// TIA Portal project "TP2 [A2182]" (V20)

(* hardware
DEVICE "S7-1200 station_1"  S7-1200 Station
   slot 0: "Rack_0"  S7-1200 Rack  Rack  V1.0
   slot 1: "PLC_1"  CPU 1215C DC/DC/Rly  6ES7 215-1HG40-0XB0  V4.2
DEVICE "SINAMICS G_1"  Sinamics.Device
   slot 0: "	_0"  Rail  SinamicsG120SVecto
   slot 0: "Drive_1"  G120 CU250S-2 PN Vector  6SL3246-0BA22-1FA0  4.7.6
      slot 1: "PROFINET interface"  MDD-SinamicsG120-P
   slot 3: "PM240-2 IP20"  PM240-2 IP20  6SL3210-1PB13-8ULx  -
DEVICE "HMI_1"  KTP700 Basic PN
   slot 0: "HMI_1"  KTP700 Basic PN  6AV2 123-2GB03-0AX0  17.0.0.0
   slot 1: "HMI_RT_1"  KTP700 Basic PN  6AV2 123-2GB03-0AX0  17.0.0.0
   slot 5: "HMI_1.IE_CP_1"  PROFINET Interface  17.0.0.0
      slot 1: "PROFINET Interface_1"  PROFINET Interface
         slot 1: "Port_1"  Port
*)

// ===== PLC "PLC_1"  CPU 1215C DC/DC/Rly =====

VAR_GLOBAL   // PLC tag table "Variateur"
   "Ix_EquartVitesse" AT %I500.0 : Bool;   // True = Dans la tolérance, OK
   "Ix_CommandeDemandé" AT %I500.1 : Bool;   // True = OK
   "Ix_VitesseAtteinte" AT %I500.2 : Bool;   // True = Atteint
   "Ix_LimiteCouple" AT %I500.3 : Bool;   // True = Couple Atteint
   "Ix_Frein" AT %I500.4 : Bool;   // True =Freiné
   "Ix_AlarmeSurchauffe" AT %I500.5 : Bool;   // True = OK
   "Ix_RotationDroite" AT %I500.6 : Bool;   // True = Droite
   "Ix_SurchauffeVariateur" AT %I500.7 : Bool;   // True = OK
   "Ix_PretEnclanchement" AT %I501.0 : Bool;   // True = Pret
   "Ix_MoteurTourne" AT %I501.1 : Bool;   // True = Moteur ON
   "Ix_FonctionnementDébloqué" AT %I501.2 : Bool;   // True = OK
   "Ix_DéfautActif" AT %I501.3 : Bool;   // True = Défauts
   "Ix_Arret2innactif" AT %I501.4 : Bool;   // True = Désactivé
   "Ix_Arret3innactif" AT %I501.5 : Bool;   // True = Désactivé
   "Ix_BloquageActif" AT %I501.6 : Bool;   // True = Bloqué
   "Ix_AlarmesActives" AT %I501.7 : Bool;   // True = Actif
   "Iw_Consigne" AT %IW502 : Int;
   "Qx_PilotageParCPU" AT %Q500.2 : Bool;   // Mettre à true
   "Qx_MarcheArret1" AT %Q501.0 : Bool;   // Mettre à true
   "Qx_MarcheArret2" AT %Q501.1 : Bool;   // Mettre à true
   "Qx_ArretRapide" AT %Q501.2 : Bool;   // Mettre à true
   "Qx_DébloquerVariateur" AT %Q501.3 : Bool;   // Mettre à true
   "Qx_BloquageRampe" AT %Q501.4 : Bool;   // Mettre à true
   "Qx_DébloquerRampe" AT %Q501.5 : Bool;   // Mettre à true
   "Qx_DébloquerConsigne" AT %Q501.6 : Bool;   // Mettre à true
   "Qx_AcquiterDéfauts" AT %Q501.7 : Bool;   // Passage de 0 à 1
   "Qw_Consigne" AT %QW502 : Int;
END_VAR

DATA_BLOCK "DB_HMI"   // DB1
{ S7_Optimized_Access := 'TRUE' }
VERSION : 0.1
   VAR
      G120 : Struct
         ActVelocity : Real;   // Vitesse actuelle (sortie bloc)
         SpeedSp : Real;   // Consigne vitesse (entrée bloc)
         RefSpeed : Real;   // Vitesse référence
         EnableAxis : Bool;   // Démarrage moteur
         AckError : Bool;   // Acquittement défaut
         StatusWord : Struct
            AxisEnabled : Bool;   // Moteur activé (sortie)
            Error : Bool;   // Défaut présent (sortie)
            Lockout : Bool;   // Verrouillage (sortie)
         END_STRUCT;
      END_STRUCT;
   END_VAR
BEGIN
END_DATA_BLOCK

FUNCTION "Block_1" : Void   // FC1, LAD
{ S7_Optimized_Access := 'TRUE' }
VERSION : 0.1
BEGIN
END_FUNCTION

ORGANIZATION_BLOCK "Main"   // OB1, LAD, ProgramCycle
TITLE = "Main Program Sweep (Cycle)"
{ S7_Optimized_Access := 'TRUE' }
VERSION : 0.1
   VAR_INPUT
      Initial_Call : Bool;   // Initial call of this OB
      Remanence : Bool;   // =True, if remanent data are available
   END_VAR
BEGIN

REGION Network 1
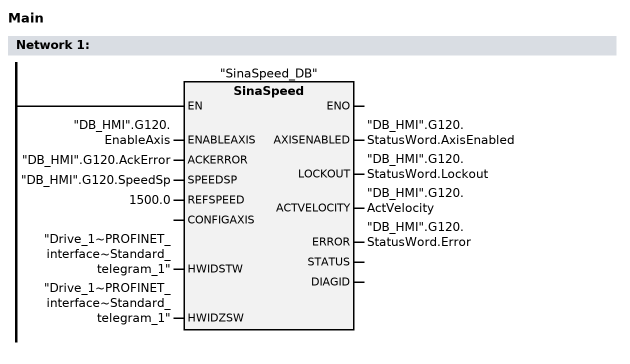
   "SinaSpeed_DB"(EnableAxis := "DB_HMI".G120.EnableAxis,   // SinaSpeed
                  AckError := "DB_HMI".G120.AckError,
                  SpeedSp := "DB_HMI".G120.SpeedSp,
                  RefSpeed := 1500.0,
                  HWIDSTW := "Drive_1~PROFINET_interface~Standard_telegram_1",
                  HWIDZSW := "Drive_1~PROFINET_interface~Standard_telegram_1",
                  AxisEnabled => "DB_HMI".G120.StatusWord.AxisEnabled,
                  Lockout => "DB_HMI".G120.StatusWord.Lockout,
                  ActVelocity => "DB_HMI".G120.ActVelocity,
                  Error => "DB_HMI".G120.StatusWord.Error);
END_REGION
END_ORGANIZATION_BLOCK

(* ===== HMI "HMI_RT_1" =====
system functions are stored by id; their names below are inferred from use
connection "HMI_Connection_1": ETHERNET, SMART_S7_1200_OMS

HMI tags "Default tag table"
   "Tag_ScreenNumber" : UInt, internal
   "DB_HMI_G120_SpeedSp" : Real = PLC DB_HMI.G120.SpeedSp, 1 s
   "DB_HMI_G120_ActVelocity" : Real = PLC DB_HMI.G120.ActVelocity, 1 s
   "DB_HMI_G120_StatusWord_AxisEnabled" : Bool = PLC DB_HMI.G120.StatusWord.AxisEnabled, 1 s
   "DB_HMI_G120_StatusWord_Error" : Bool = PLC DB_HMI.G120.StatusWord.Error, 1 s
   "DB_HMI_G120_EnableAxis" : Bool = PLC DB_HMI.G120.EnableAxis, 1 s
   "DB_HMI_G120_AckError" : Bool = PLC DB_HMI.G120.AckError, 1 s

Template "Template_1" 800x480
   Button "Exit" at 714,429 size 71x50; TextOff 'Exit'; PictureOff "ExitRuntime_KTP700_Basic_PN_TR"; PictureOn "ExitRuntime_KTP700_Basic_PN_TR"
      on Release: StopRuntime(0)
   Button "Template_Button" at 614,429 size 71x50; TextOff 'Text'
   Button "Template_Button_1" at 514,429 size 71x50; TextOff 'Text'
   Button "Template_Button_2" at 414,429 size 71x50; TextOff 'Text'
   Button "Template_Button_3" at 314,429 size 71x50; TextOff 'Text'
   Button "Template_Button_4" at 214,429 size 71x50; TextOff 'Text'
   Button "Alarms" at 114,429 size 71x50; TextOff 'Alarms'; PictureOff "AlarmDisplay_KTP700_Basic_PN_TR"; PictureOn "AlarmDisplay_KTP700_Basic_PN_TR"
      on Release: function_ef3f5d25("Alarm window_Unacknowledged", -1)
   Button "Start screen" at 14,429 size 71x50; TextOff 'Start screen'; PictureOff "NavigateHome_KTP700_Basic_PN_TR"; PictureOn "NavigateHome_KTP700_Basic_PN_TR"
      on Release: ActivateScreen("Root screen", 0)
   SymbolicIOField "Symbolic_IO_Field_Screen" at 93,9 size 600x33; TextOff '0'; TextOn '1'; TextList "TextList_ScreenNames"
      ProcessValue <- "Tag_ScreenNumber"
      on Change: ActivateScreenByNumber("Tag_ScreenNumber", 0)
   DateTimeField "HmiScreenItemData" at 695,25 size 105x25
   DateTimeField "HmiScreenItemData_1" at 695,0 size 105x25
   GraphicView "Logo" at 0,0 size 91x51; Picture "Logo of HMI_1"

screen "Root screen" 800x480, template "Template_1"
   on GenerateScreen: SetTag("Tag_ScreenNumber", 1)
   Button "Button_1" at 415,178 size 96x32; TextOff 'AckError'
      on Press: SetBit("DB_HMI_G120_AckError")
   Button "Button_2" at 278,178 size 96x32; TextOff 'EnableAxis'
      on Press: SetBit("DB_HMI_G120_EnableAxis")
   Button "Button_3" at 343,224 size 96x32; TextOff 'HALT'
      on Press: ResetBit("DB_HMI_G120_EnableAxis")
   IOField "I/O field_1" at 426,93 size 96x32; FormatPattern 9999
      ProcessValue <- "DB_HMI_G120_SpeedSp"
   Rectangle "Rectangle_1" at 276,115 size 30x30
      Appearance <- "DB_HMI_G120_StatusWord_AxisEnabled"
   Bar "Bar_1" at 257,299 size 324x80; MinimumValue 0; MaximumValue 1500
      ProcessValue <- "DB_HMI_G120_ActVelocity"
   Rectangle "Rectangle_2" at 323,115 size 30x30
      Appearance <- "DB_HMI_G120_StatusWord_Error"
   TextField "Text field_2" at 275,146 size 39x23; Text 'ENA'
   TextField "Text field_3" at 323,146 size 39x23; Text 'ERR'
   TextField "Text field_4" at 267,94 size 148x23; Text 'Velocity set rpm :'
   TextField "Text field_1" at 257,269 size 173x23; Text 'Actual velocity rpm :'
*)